// SIMATIC S7-200 SMART project (STEP 7-Micro/WIN SMART), CPU ST60

ORGANIZATION_BLOCK MAIN:OB1
TITLE=程序注释
BEGIN
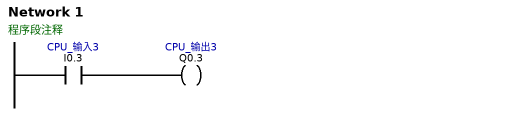
Network 1
// 程序段注释
LD     CPU_输入3:I0.3
=      CPU_输出3:Q0.3
END_ORGANIZATION_BLOCK
